{attribute 'GeneratedUsingTerminal: EL2258-0000-0017'}
{attribute addProperty BoxType "EL2258-0000-0017"}
{attribute addProperty Id "Output_short_circuitBOOL1Output_buffer_overflowBOOL1Output_stateBOOL1Input_cycle_counterBYTE1Output_order_feedbackUSINT1Events_in_output_bufferUSINT1"}
{attribute addProperty CRC "1680617169"}
{attribute addProperty Size "6"}
TYPE Status_642C2ED1 :
STRUCT
	{attribute addProperty Name "Output_short_circuit"}
	Output_short_circuit : BOOL;
	{attribute addProperty Name "Output_buffer_overflow"}
	Output_buffer_overflow : BOOL;
	{attribute addProperty Name "Output_state"}
	Output_state : BOOL;
	{attribute addProperty Name "Input_cycle_counter"}
	Input_cycle_counter : BYTE;
	{attribute addProperty Name "Output_order_feedback"}
	Output_order_feedback : USINT;
	{attribute addProperty Name "Events_in_output_buffer"}
	Events_in_output_buffer : USINT;
END_STRUCT
END_TYPE

(* stored: Version 1.2.0.0, ProductVersion 3.1.4024.11
   DUT Status_642C2ED1: Id {46b900b0-8ac1-4dd0-bc09-3bd1d77cd6a2} *)
